// TIA Portal V18 export
FUNCTION "Interlock" : Void   // FC1, F_LAD
{ S7_Optimized_Access := 'TRUE' }
VERSION : 0.1
// stored: AutoNumber true, IsIECCheckEnabled false, UDAEnableTagReadback false
   VAR_INPUT
      Room1_Interlock : Bool;
      Room2_Interlock : Bool;
      ACC_Interlock : Bool;
      VerticalBeam_Interlock : Bool;
      "E-stop" : Bool;
   END_VAR
BEGIN

REGION Network 1
   // 暂未考虑模块钝化和通道钝化情况
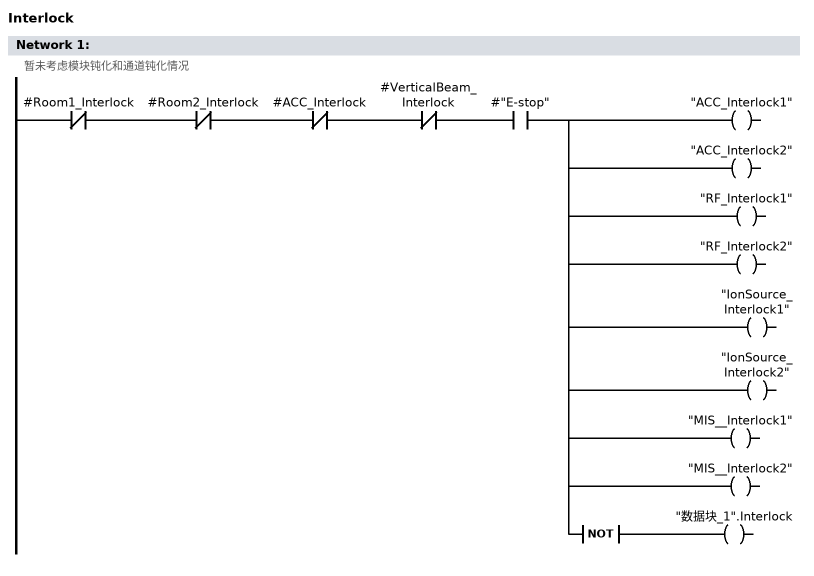
   RUNG wire#powerrail
      I_Contact( #Room1_Interlock )
      I_Contact( #Room2_Interlock )
      I_Contact( #ACC_Interlock )
      I_Contact( #VerticalBeam_Interlock )
      Contact( #"E-stop" )
      wire#w1
      Coil( "ACC_Interlock1" )
   END_RUNG
   RUNG wire#w1
      Coil( "ACC_Interlock2" )
   END_RUNG
   RUNG wire#w1
      Coil( "RF_Interlock1" )
   END_RUNG
   RUNG wire#w1
      Coil( "RF_Interlock2" )
   END_RUNG
   RUNG wire#w1
      Coil( "IonSource_Interlock1" )
   END_RUNG
   RUNG wire#w1
      Coil( "IonSource_Interlock2" )
   END_RUNG
   RUNG wire#w1
      Coil( "MIS__Interlock1" )
   END_RUNG
   RUNG wire#w1
      Coil( "MIS__Interlock2" )
   END_RUNG
   RUNG wire#w1
      Not()
      Coil( "数据块_1".Interlock )
   END_RUNG
   // the same network as SCL:
   "ACC_Interlock1" := NOT #Room1_Interlock AND NOT #Room2_Interlock AND NOT #ACC_Interlock AND NOT #VerticalBeam_Interlock AND #"E-stop";
   "ACC_Interlock2" := "ACC_Interlock1";
   "RF_Interlock1" := "ACC_Interlock1";
   "RF_Interlock2" := "ACC_Interlock1";
   "IonSource_Interlock1" := "ACC_Interlock1";
   "IonSource_Interlock2" := "ACC_Interlock1";
   "MIS__Interlock1" := "ACC_Interlock1";
   "MIS__Interlock2" := "ACC_Interlock1";
   "数据块_1".Interlock := NOT "ACC_Interlock1";
END_REGION
END_FUNCTION
